# B&R Automation Studio project Guziczki_i_swiatelka
Automation Studio 4.9

## Configuration Config1

### Task classes (Cpu.sw)
```
Cyclic#4 (cycle 100000 us, tolerance 100000 us):
  Program1 <- Program1.prg
Libraries: standard
```

### Hardware
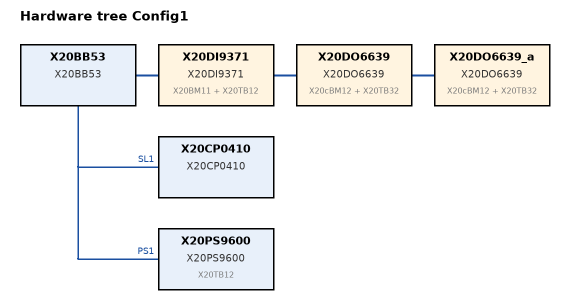
```
X20BB53 : X20BB53 v1.0.1.0
X20BM11 : X20BM11 v1.1.0.0  [X2X1 -> X20BB53.IF6]
X20CP0410 : X20CP0410 v1.7.3.0  [SL -> X20BB53.SL1]
  Connector IF2:
    ActivateDevice = 1
    Mode = Manual
    InternetAddress = 192.168.0.1
    SubnetMask = 255.255.255.0
  ConfigurationID = Guziczki_i_swiatelka_Config1
  TimerDeviceType = SWIOTIMER
  Cyclic1Duration = 10000
  Cyclic1Tolerance = 10000
  Cyclic2Duration = 20000
  Cyclic2Tolerance = 20000
  Cyclic3Duration = 50000
  Cyclic3Tolerance = 50000
  Cyclic4Duration = 100000
  Cyclic4Tolerance = 100000
  Cyclic5Duration = 200000
  Cyclic5Tolerance = 200000
  Cyclic6Duration = 500000
  Cyclic6Tolerance = 500000
  Cyclic7Duration = 1000000
  Cyclic7Tolerance = 1000000
  Cyclic8Duration = 10000
  Cyclic8Tolerance = 30000000
  FileDevice1
  FileDeviceName1 = USER
  FileDevicePath1 = USER_PATH
X20DI9371 : X20DI9371 v1.6.1.0  [SS1 -> X20TB12_a.SS; SL -> X20BM11.SL1]
X20DO6639 : X20DO6639 v1.2.2.0  [SS1 -> X20TB32.SS; SL -> X20cBM12.SL1]
X20DO6639_a : X20DO6639 v1.2.2.0  [SS1 -> X20TB32_a.SS; SL -> X20cBM12_a.SL1]
  Supervision = off
X20PS9600 : X20PS9600 v1.6.2.0  [PS -> X20BB53.PS1; SS1 -> X20TB12.SS]
X20TB12 : X20TB12 v1.0.0.0
X20TB12_a : X20TB12 v1.0.0.0
X20TB32 : X20TB32 v1.0.0.1
X20TB32_a : X20TB32 v1.0.0.1
X20cBM12 : X20cBM12 v1.1.0.0  [X2X1 -> X20BM11.X2X2]
X20cBM12_a : X20cBM12 v1.1.0.0  [X2X1 -> X20cBM12.X2X2]
```

### IoMap.iom - X20CP0410/IoMap.iom
```iecst
VAR_CONFIG
	::input_1 AT %IX."X20DI9371".DigitalInput01;
	::input_2 AT %IX."X20DI9371".DigitalInput02;
	output_1  AT %QX."X20cDO6639".DigitalOutput01;
	output_2 AT %QX."X20cDO6639".DigitalOutput02;
	output_3 AT %QX."X20cDO6639".DigitalOutput03;
	output_4  AT %QX."X20cDO6639".DigitalOutput04;
	output_5 AT %QX."X20cDO6639".DigitalOutput05;
	output_6  AT %QX."X20cDO6639".DigitalOutput06;
END_VAR
```

## Logical view

### Global.var - Global variables
```iecst
VAR
	input_1 : BOOL;
	input_2 : BOOL;
	output_1 : BOOL;
	output_2 : BOOL;
	output_3 : BOOL;
	output_4 : BOOL;
	output_5 : BOOL;
	output_6 : BOOL;
END_VAR
```

### Program Logical/Program1 (IEC)

#### Main.st - Init, cyclic, exit code
```iecst
PROGRAM _INIT
	delay_1(IN :=start_delay,PT := T#1s,Q :=output_1);
	delay_2(IN :=output_1,PT := T#1s,Q :=output_2);
	delay_3(IN :=output_2,PT := T#1s,Q :=output_3);
	delay_4(IN :=output_3,PT := T#1s,Q :=output_4);
	delay_5(IN :=output_4,PT := T#1s,Q :=output_5);
	delay_6(IN :=output_5,PT := T#1s,Q :=output_6);

END_PROGRAM

PROGRAM _CYCLIC
	IF input_1 AND input_2 THEN

		start_delay := TRUE;
	END_IF

END_PROGRAM

PROGRAM _EXIT
	(* Insert code here *)

END_PROGRAM
```

#### Variables.var - Local variables
```iecst
VAR
	delay_1 : TON;
	delay_2 : TON;
	delay_3 : TON;
	delay_4 : TON;
	delay_5 : TON;
	delay_6 : TON;
	start_delay : BOOL;
	end_delay : BOOL;
END_VAR
```

#### LocalFunctions.fun
```iecst
{REDUND_ERROR} {REDUND_UNREPLICABLE} FUNCTION_BLOCK PWM (*TODO: Add your comment here*) (*$GROUP=User,$CAT=User,$GROUPICON=User.png,$CATICON=User.png*)
	VAR_INPUT
		duty_cycle :  REAL;
		period :  TIME := T#1s;
		input_PWM : BOOL;
	END_VAR

	VAR

		time_on : TIME;
		time_off : TIME;
		timer_on : TON;
		timer_off : TON;

	END_VAR

	VAR_OUTPUT
	out: BOOL;
	END_VAR

END_FUNCTION_BLOCK
```

#### PWM.st
```iecst
(* TODO: Add your comment here *)
FUNCTION_BLOCK PWM
(*Obliczenie czsów*)
	time_on := REAL_TO_TIME(TIME_TO_REAL(period)*(duty_cycle/100));
	time_off := ABS(INT_TO_TIME(REAL_TO_INT(duty_cycle)- TIME_TO_INT(time_on)));
	(*timery sterujace opuźnionym włączeniem i wyłączeniem PWM*)
	timer_off(IN:=input_PWM AND NOT timer_on.Q,PT:=time_off);
	timer_on(IN:=input_PWM AND timer_off.Q,PT:=time_on);

	IF input_PWM THEN
		IF duty_cycle <=0 THEN
			out := FALSE;
		ELSIF duty_cycle >= 100 THEN
			out := TRUE;
		ELSE
			out := timer_off.Q;
		END_IF
	ELSE
		out := FALSE;
	END_IF
END_FUNCTION_BLOCK
```

#### Cyclic.st
```iecst
PROGRAM _CYCLIC
	PWM_1(duty_cycle :=30, period :=T#1s , input_PWM :=input_3 );
IF PWM_1.out THEN
	output_5 := TRUE;
	output_6 := TRUE;
ELSE
	(* statements if false *)
END_IF;

END_PROGRAM
```

Listed in the project but not available here: Logical/Global.typ, Logical/Libraries, Logical/Program1/Types.typ
